{attribute 'qualified_only'}
{attribute 'strict'}
{attribute 'to_string'}
TYPE E_INSTANCE_STATE :
(
	INVALID,
  INIT,
  DISABLED,
  DETECT_IN_LIST,
  ENABLED,
  WORKING,
  FINISH
);
END_TYPE

(* stored: Version 1.1.0.1, ProductVersion 3.1.4024.13
   DUT E_INSTANCE_STATE: Id {54ac76f8-93e6-4095-9fff-f1c1dcff5aa1} *)
